///Automatically created by BoxConfigurator
VAR_GLOBAL
END_VAR

(* stored: Version 1.1.0.1, ProductVersion 3.1.4024.9
   GVL GVL_Safety: Id {20e96d49-2f70-454f-bddd-8993744cbceb} *)
